FUNCTION_BLOCK CLIENT_m_n_TEST (* Test CLIENT_m_n in a Composite Function Block *)
  (* Standard: 61499-2 *)
  (* Version 0.0, 2002-12-17, JHC, Rockwell Automation *)
  (* Compiler header: package fb.rt.test; import fb.rt.net.*; *)
  (* Compiler Java IBM Jikes 1.06 *)
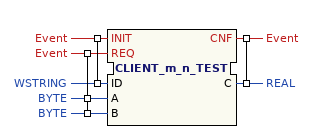
  EVENT_INPUT
    INIT WITH ID;
    REQ WITH A, B; (* Normal Execution Request *)
  END_EVENT
  EVENT_OUTPUT
    CNF WITH C; (* Execution Confirmation *)
  END_EVENT
  VAR_INPUT
    ID : WSTRING;
    A : BYTE;
    B : BYTE;
  END_VAR
  VAR_OUTPUT
    C : REAL;
  END_VAR
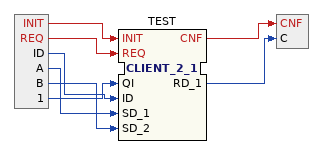
  FBS
    TEST : CLIENT_2_1;
  END_FBS
  EVENT_CONNECTIONS
    INIT TO TEST.INIT;
    REQ TO TEST.REQ;
    TEST.CNF TO CNF;
  END_CONNECTIONS
  DATA_CONNECTIONS
    1 TO TEST.QI;
    ID TO TEST.ID;
    A TO TEST.SD_1;
    B TO TEST.SD_2;
    TEST.RD_1 TO C;
  END_CONNECTIONS
END_FUNCTION_BLOCK
